// TIA Portal project "Project_IOLINKSafety" (V18)

(* hardware
DEVICE "S7-1200 station_1"  S7-1200 Station
   slot 0: "Rack_0"  S7-1200 Rack  Rack  V1.0
   slot 1: "PLC_1"  CPU 1212FC DC/DC/DC  6ES7 212-1AF40-0XB0  V4.6
DEVICE "GSD device_1"  GSD.Device.PN
   slot 0: "Rack"  Rack  V1.0
   slot 0: "AXL-F-BK-PN-TPS"  AXL F BK PN TPS  2403869  1.32
      slot 0: "AXL F BK PN TPS"  AXL F BK PN TPS
      slot 1: "Interface"  Interface
         slot 1: "RJ45 10/100 MBit/s"  RJ45 10/100 MBit/s
         slot 2: "RJ45 10/100 MBit/s_1"  RJ45 10/100 MBit/s
   slot 1: "AXL SE DI16/1_1"  AXL SE DI16/1  1088127  1.0
      slot 0: "AXL SE DI16/1"  AXL SE DI16/1
   slot 1: "Digital Input"  Digital Input
   slot 1: "AXL E IOL SDI8 SDO4 2A M12 6P PS2.4"  AXL E IOL SDI8 SDO4 2A M12 6P PS2.4
   slot 1: "AXL E IOL SDI8 SDO4 2A M12 L PS2.6"  AXL E IOL SDI8 SDO4 2A M12 L PS2.6
   slot 2: "AXL SE DO16/1_1"  AXL SE DO16/1  1088129  1.0
      slot 0: "AXL SE DO16/1"  AXL SE DO16/1
   slot 2: "Digital Input_1"  Digital Input
   slot 2: "Digital Input_1"  Digital Input
   slot 2: "Inactive_1"  Inactive
   slot 3: "AXL SE AI4 U 0-10_1"  AXL SE AI4 U 0-10  1088104  1.0
      slot 0: "AXL SE AI4 U 0-10"  AXL SE AI4 U 0-10
   slot 3: "Digital Input_2"  Digital Input
   slot 3: "Digital Input_2"  Digital Input
   slot 3: "Inactive"  Inactive
   slot 4: "AXL SE IOL4_1"  AXL SE IOL4  1088132  1.0
      slot 0: "AXL SE IOL4"  AXL SE IOL4
   slot 4: "Digital Input_3"  Digital Input
   slot 4: "Digital Input_3"  Digital Input
   slot 4: "Inactive_2"  Inactive
   slot 5: "Digital Input_4"  Digital Input
   slot 5: "Digital Input_4"  Digital Input
   slot 6: "Digital Input_5"  Digital Input
   slot 6: "Digital Input_5"  Digital Input
   slot 7: "Digital Input_6"  Digital Input
   slot 7: "Digital Input_6"  Digital Input
   slot 8: "Digital Input_7"  Digital Input
   slot 8: "Digital Input_7"  Digital Input
DEVICE "GSD device_2"  GSD.Device.PN
   slot 0: "Rack"  Rack  V1.0
   slot 0: "AXL-F-BK-PN-TPS_1"  AXL F BK PN TPS  2403869  1.32
      slot 0: "AXL F BK PN TPS"  AXL F BK PN TPS
      slot 1: "Interface"  Interface
         slot 1: "RJ45 10/100 MBit/s"  RJ45 10/100 MBit/s
         slot 2: "RJ45 10/100 MBit/s_1"  RJ45 10/100 MBit/s
   slot 1: "AXL SE DI16/1_1"  AXL SE DI16/1  1088127  1.0
      slot 0: "AXL SE DI16/1"  AXL SE DI16/1
   slot 1: "AXL E IOL SDI8 SDO4 2A M12 L PS2.6"  AXL E IOL SDI8 SDO4 2A M12 L PS2.6
   slot 2: "AXL SE DO16/1_1"  AXL SE DO16/1  1088129  1.0
      slot 0: "AXL SE DO16/1"  AXL SE DO16/1
   slot 2: "Digital Input"  Digital Input
   slot 3: "AXL SE AI4 U 0-10_1"  AXL SE AI4 U 0-10  1088104  1.0
      slot 0: "AXL SE AI4 U 0-10"  AXL SE AI4 U 0-10
   slot 3: "Digital Input_1"  Digital Input
   slot 4: "AXL SE IOL4_1"  AXL SE IOL4  1088132  1.0
      slot 0: "AXL SE IOL4"  AXL SE IOL4
   slot 4: "Digital Input_2"  Digital Input
*)

// ===== PLC "PLC_1"  CPU 1212FC DC/DC/DC =====
// protected blocks, not shown: "PRSF_AXL_E", "PRSF_DiagHandler", "PRSF_IOLM_Diag"

VAR_GLOBAL   // PLC tag table "Default tag table"
   "xActivate" AT %M0.0 : Bool;
   "Tag_1" AT %MW10 : Word;
   "Tag_2" AT %M0.1 : Bool;
   "Tag_3" AT %M0.2 : Bool;
   "Tag_4" AT %M0.3 : Bool;
   "mReset" AT %M1.3 : Bool;
   "Tag_6" AT %IW3 : Word;
   "Tag_7" AT %IW4 : Word;
   "Tag_8" AT %IW5 : Word;
   "Tag_9" AT %IW6 : Word;
   "Tag_10" AT %IW7 : Word;
   "Tag_11" AT %IW8 : Word;
   "Tag_12" AT %IW9 : Word;
   "Tag_13" AT %IW10 : Word;
   "Tag_14" AT %M1.4 : Bool;
   "siESTOP" AT %I3.0 : Bool;
   "sqESTOP1_Q" AT %Q3.0 : Bool;
END_VAR

TYPE "PRSF_UDT_IOCALL"
VERSION : 0.1
   STRUCT
      xReq : Bool;
      wHWAddr : Word;
      diCAP : DInt;
      xRDWR : Bool;
      iPort : Int;
      iIndex : Int;
      iSubindex : Int;
      iLen : Int;
      arr_b_IOLData : Array[0..231] of Byte;
      xDone_Valid : Bool;
      xBusy : Bool;
      xError : Bool;
      dwStatus : DWord;
      dwIOL_Status : DWord;
      iRD_Len : Int;
   END_STRUCT;
END_TYPE

TYPE "PRSF_UDT_DIAG"
VERSION : 0.1
   STRUCT
      wDiagCode : Word;
      wAddDiagCode : Word;
      xError : Bool;
      iState : Int;
      IOL_CallDiag : "PRSF_UDT_IOCALL";
   END_STRUCT;
END_TYPE

TYPE "PRSF_UDT_COM"
VERSION : 0.1
   STRUCT
      arr_i_Com : Array[0..255] of UInt;
      arr_HW : Array[0..8] of HW_ANY;
      arr_HW_Diag : Array[0..8] of Bool;
   END_STRUCT;
END_TYPE

DATA_BLOCK "Main_Safety_RTG1_DB"   // DB1, F_DB
{ S7_Optimized_Access := 'TRUE' }
NAME : FUSI
VERSION : 0.1
// stored: InstanceOfName Main_Safety_RTG1
"Main_Safety_RTG1"
BEGIN
END_DATA_BLOCK

DATA_BLOCK "PRSF_AXLE_UserDB"   // DB2
{ S7_Optimized_Access := 'TRUE' }
VERSION : 0.1
   VAR
      xActivate : Bool;
   END_VAR
   VAR RETAIN
      iPort : Int;
      IOLD_HWAddr : Hw_Any;
      IOLM_HWAddr : Hw_Any;
   END_VAR
   VAR
      wFAddr : Word;
      xSetFAddr : Bool;
      xErrorAck : Bool;
      wDevFAddr : Word;
      strDevSerial : String[13];
      xDiagAvailable : Bool;
      stDiagState : Struct
         uiLfdNo : UInt;
         uiPrio : UInt;
         bChannel : Byte;
         wCode : Word;
         FunctionGorup : String[8];
         dwAddValue : DWord;
         uiTextLength : UInt;
         strText : String[100];
      END_STRUCT;
      udtDiag : "PRSF_UDT_DIAG";
   END_VAR
BEGIN
END_DATA_BLOCK

DATA_BLOCK "Data_block_1"   // DB6
{ S7_Optimized_Access := 'TRUE' }
VERSION : 0.1
   VAR
      bytes : Array[0..999] of Byte;
   END_VAR
BEGIN
END_DATA_BLOCK

DATA_BLOCK "PRSF_AXL_E_COM"   // DB3200
{ S7_Optimized_Access := 'TRUE' }
VERSION : 0.1
   VAR
      udtCom : "PRSF_UDT_COM";
   END_VAR
BEGIN
END_DATA_BLOCK

FUNCTION_BLOCK "Main_Safety_RTG1"   // FB1, F_FBD
{ S7_Optimized_Access := 'TRUE' }
   VAR
      ACK_GL_Instance : ACK_GL;
      ESTOP1 : ESTOP1;
   END_VAR
   VAR CONSTANT
      OFF : Bool;
      ON : Bool := 1;
   END_VAR
BEGIN

REGION Network 1
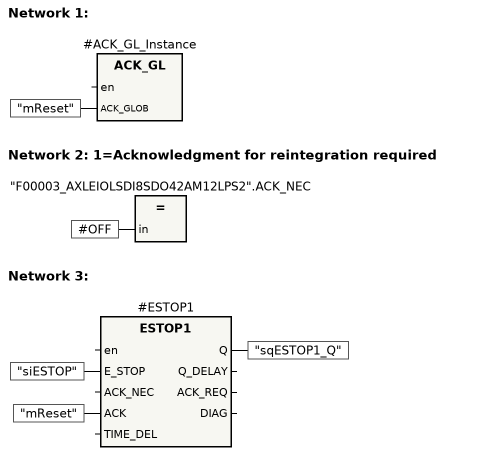
   #ACK_GL_Instance(ACK_GLOB := "mReset");   // ACK_GL
END_REGION

REGION Network 2: 1=Acknowledgment for reintegration required
   "F00003_AXLEIOLSDI8SDO42AM12LPS2".ACK_NEC := #OFF;
END_REGION

REGION Network 3
   #ESTOP1(E_STOP := "siESTOP", ACK := "mReset", Q => "sqESTOP1_Q");   // ESTOP1
END_REGION
END_FUNCTION_BLOCK

FUNCTION_BLOCK "IO_LINK_DEVICE"   // FB50001, SCL
TITLE = IO_LINK_DEVICE
{ S7_Optimized_Access := 'TRUE' }
AUTHOR : SUP_FA
FAMILY : IO-Link
VERSION : 3.0
// Function block to read and write acyclic data on devices with IO-Link used on SIMATIC S7 controllers. (former IO_LINK_CALL)
   VAR_INPUT
      REQ : Bool;   // Request Function / Neuer Auftrag / request function
      ID : Hw_Io;   // Hardwarekennung des IOL-Master Moduls (HW_IO) aus HW-Konfiguration / hardware identifier of IO-Link master module (HW_IO) from hw-config
      CAP : DInt := DINT#0;   // Client Access Point (CAP), bei ET200 immer 227 dez / Client Access Point (CAP), for ET200 always 227 decimal
      RD_WR : Bool;   // Lese und Schreibzugriff auf IO-Link Device 0: Lesen, 1: schreiben / read and write access on IO-Link device 0: read, 1: write
      PORT : Int := INT#0;   // Port/ Kanalnummer an dem das IO-Link Device betrieben wird. (ET200 = 0 .. 4) / number of port on IO-Link master module (ET200SP = 0..4)
      IOL_INDEX : Int := INT#0;   // Adressparameter Index (IO-Link Device) 0..32767 IOL-D, 65535 port functions / address parameter Index (IO-Link Device) 0..32767 IOL-D, 65535 port functions
      IOL_SUBINDEX : Int := INT#0;   // Adressparameter Subindex (IO-Link Device) 0 ges. Record; 1-255 einz. Parameter / address parameter Subindex (IO-Link Device) 0 full record; 1-255 single parameter
      LEN : Int := INT#0;   // Länge der zu schreibenden Daten (Nettodaten) / length of writing data (netto data)
   END_VAR
   VAR_OUTPUT
      DONE_VALID : Bool;   // Gültigkeit 0: Daten nicht gültig; 1: Daten gültig / validity 0: data invalid ; 1: data valid
      BUSY : Bool;   // 0: Auftrag abgeschlossen 1: Auftrag in Bearbeitung / 0: request finish 1: request in progress
      ERROR : Bool;   // Fehler Flag 0: kein Fehler; 1: Abbruch der Funktion mit Fehler / Error Flag = 0: no error; 1: function aborted with error
      STATUS : DWord := DW#16#00000000;   // DP/ PNIO - Fehlerstatus; ERROR Flag = 1 - detaillierter Kommunikationsfehlerstatus / DP/ PNIO - error status ; ERROR Flag = 1 - communication error status in detail
      IOL_STATUS : DWord := DW#16#00000000;   // IO-Link Fehlerstatus; ERROR Flag = 1 - detaillierte IO-Link Fehlerstatus / IO-Link error status; ERROR flag = 1: IO-Link error status in detail
      RD_LEN : Int := INT#0;   // Länge des gelesenen Datensatzes (Anzahl Bytes) / length of read data record (number of bytes)
   END_VAR
   VAR_IN_OUT
      RECORD_IOL_DATA : Array[0..231] of Byte;   // Datenbereich für LESEN / SCHREIBEN (max. 232 Byte) / data area for reading / writing data (max. 232 byte)
   END_VAR
   VAR
      RDREC_Function : RDREC;   // Funktion Datensatz lesen (ehemals SFB52) / system function "read data record" (former SFB52)
      WRREC_Function : WRREC;   // Funktion Datensatz schreiben (ehemals SFB53) / system function "write data record" (former SFB53)
      TP_poll : TP_TIME;   // Pollzeit für "Datensatz lesen" / poll rate read data record
      TON_monitoring : TON_TIME;   // Überwachungszeit für Aufträge / request monitoring time
      rdrec : Struct   // interne Struktur für RDREC / internal structure for RDREC
         valid : Bool;   // Function performed
         busy : Bool;   // Function busy
         error : Bool;   // Error flag
         status : DWord;   // Function result/error message
         length : UInt;   // Length of the fetched data record
      END_STRUCT;
      wrrec : Struct   // interne Struktur für WRREC / internal structure for WRREC
         length : UInt;   // length of write data record
         done : Bool;   // Function performed
         busy : Bool;   // Function busy
         error : Bool;   // Error flag
         status : DWord;   // Function result/error message
      END_STRUCT;
      read : Struct   // Datenbereich für Lesedaten / data area for reading data
         header : Struct
            CALL : Struct   // header for read/write data record
               Extended_Function_Num : Byte := 16#8;   // extended function number (fix coded 08h)
               Port : Byte;   // variable port (user interface) 0...255
               FI_Index : Word := 16#FE4A;   // FI index (fix coded 65098)
            END_STRUCT;
            IOL : Struct   // header for IO-Link
               Control : Byte;   // RD_WR = 0 = read = Control:=0x03 / / RD_WR = 1 = write = Control:=0x02
               Index_HighByte : Byte;   // index of data record 0…32767 (high byte)
               Index_LowByte : Byte;   // index of data record 0…32767 (low byte)
               Subindex : Byte;   // subindex for data record 0...255
            END_STRUCT;
         END_STRUCT;
         data : Array[0..231] of Byte;
      END_STRUCT;
      write : Struct   // Datenbereich für Schreibdaten / data area for writing data
         header : Struct
            CALL : Struct   // header for read/write data record
               Extended_Function_Num : Byte := 16#8;   // extended function number (fix coded 08h)
               Port : Byte;   // variable port (user interface) 0...255
               FI_Index : Word := 16#FE4A;   // FI index (fix coded 65098)
            END_STRUCT;
            IOL : Struct   // header for IO-Link
               Control : Byte;   // RD_WR = 0 = read = Control:=0x03 / / RD_WR = 1 = write = Control:=0x02
               Index_HighByte : Byte;   // index of data record 0…32767 (high byte)
               Index_LowByte : Byte;   // index of data record 0…32767 (low byte)
               Subindex : Byte;   // subindex for data record 0...255
            END_STRUCT;
         END_STRUCT;
         data : Array[0..231] of Byte;
      END_STRUCT;
      sequencecontrol : Int := INT#0;   // number of sequence control
      typeofrequest : Int := INT#0;   // type of request (0=Read, 1=Write)
      R_TRIG_REQ : Bool;   // Impuls für neuen Auftrag starten / impulse start new request
      R_TRIG_REQ_old : Bool;   // Flankenmerker / old value of REQ (previous cycle)
      F_TRIG_poll : Bool;   // Impuls für Pollen "Datensatz lesen" / impulse poll read data record (response)
      F_TRIG_poll_old : Bool;   // Flankenmerker / old value of Poll (previous cycle)
   END_VAR
   VAR_TEMP
      retval : Int;   // Variable für Rückgabewerte von Funktionen / function return value
      tmpWORD : Word;   // Datentyp WORD zur temporären Verwendung / data type WORD for temporarily use
      tmpDWORD : DWord;   // Datentyp DWORD zur temporären Verwendung / data type DWORD for temporarily use
      tmpINT : Int;   // Datentyp INT zur temporären Verwendung / data type INT for temporarily use
      i : Int;   // Laufvariable für for-Schleifen / run tag for counting loops
   END_VAR
BEGIN
   (*---------------------------------------------------------------------------------------------------------------------
   SIEMENS AG
   ©Copyright 2015. All Rights Reserved.
   -----------------------------------------------------------------------------------------------------------------------
   Limitation of liability
   This software was developed with largest care. However, the author can not guarantee, that the software runs under
   each version of STEP7 on each PLC flawlessly.
   There is no warranty for the software, to the extent permitted by applicable law. The copyright holder provides the
   software "as is" without warranty of any kind, either expressed or implied, including, but not limited to, the implied
   warranties of merchantability and fitness for a particular purpose. The entire risk as to the quality and performance
   of the software is with you. Should the software prove defective, you assume the cost of all necessary servicing,
   repair or correction. In no event unless required by applicable law will the copyright holder be liable to you for
   damages, including any general, special, incidental or consequential damages arising out of the use or inability to
   use the software (including but not limited to loss of data or data being rendered inaccurate or losses sustained by
   you or third parties or a failure of the software to operate with any other programs), even if such holder or other
   party has been advised of the possibility of such damages.
   Permission to use or copy this software for any purpose is hereby granted without fee, provided the above notices are
   retained on all copies. Permission to modify the code and to distribute modified code is granted, provided the above
   notices are retained, and a notice that the code was modified is included with the above copyright notice.
   -----------------------------------------------------------------------------------------------------------------------
   Functionality provided by this source (short description):
   Function block IO_LINK_DEVICE - used to read and write of acyclic data records on devices with IO-Link.
   Note:
   To read data records, the IO-Link master modules needs to know which data record is required. Therefore it is necessary
   to send at first a request via write data record (only header of 8 byte). As response the IO-Link master module
   will send the required data record.

   Status:     Released (tested)
   File name:  IO_LINK_DEVICE
   System :    SIMATIC S7-1200/1500
   Version :   3.1
   -----------------------------------------------------------------------------------------------------------------------
   Script to be stored on level ... in project (mark appropriate levels with [x] below)
   [ ] External
   [ ] All levels possible
   [x] Project level
   [ ] Controller level
   [ ] Device level
   [ ] Subobject level
   -----------------------------------------------------------------------------------------------------------------------
   Restrictions, known limitations:
   The limitation of 240 byte is based on PROFIBUS DP protocol. With PROFINET IO there wouldn't no limit but because of 
   compatibility reason it wasn't changed.
     - header =   8 byte
     - data   = 232 byte
   -----------------------------------------------------------------------------------------------------------------------
   Requirements, prerequisites, External resources used: nothing
   -----------------------------------------------------------------------------------------------------------------------
   Change log table (latest change is at the bottom OF the list):
   Version Date Changes applied
   V2.0.0 <2013-09-30> First created with TIA Portal V12 SP1
   V2.1.0 <2014-03-14> Upgrade system function 'WRREC' from V1.0 to V1.1 and released for TIA Portal V13
   V3.0.0 <2015-02-28> Upgrade and released for TIA Portal V13 SP1 (without backup/restore master parameter)
   V3.1.0 <2015-09-15> Change of #IOL_INDEX and #Port lower boundry to 0 and Improved behaviour when called in cyclic OBs with > 100ms
   ---------------------------------------------------------------------------------------------------------------------*)

   (*---------------------------------------------------------------------------------------------------------------------
   Description of programmed IO-Link error codes
   8000 = time out
   8001 = wrong port
   8002 = wrong index
   8003 = wrong subindex
   8005 = wrong length for write data record
   8006 = wrong length for read data record
   8052 = error during reading data record
   8053 = error during writing data record
   All other codes are coming from a higher level!
   ---------------------------------------------------------------------------------------------------------------------*)

   (*---------------------------------------------------------------------------------------------------------------------
               NEW REQUEST
   ---------------------------------------------------------------------------------------------------------------------*)
   // detection rising edge of "REQ"
   #R_TRIG_REQ := #REQ = TRUE AND #R_TRIG_REQ_old = FALSE;
   #R_TRIG_REQ_old := #REQ = TRUE;

   // start new request if not busy
   IF #R_TRIG_REQ = TRUE AND #sequencecontrol = 0 THEN
       // Freeze record ID and CAP
       #WRREC_Function.ID := #ID;
       #WRREC_Function.INDEX := #CAP;
       #RDREC_Function.ID := #ID;
       #RDREC_Function.INDEX := #CAP;

       // Initialize outputs
       #DONE_VALID := FALSE;
       #BUSY := TRUE;
       #ERROR := FALSE;
       #STATUS := DW#16#00000000;
       #IOL_STATUS := DW#16#00000000;
       #RD_LEN := INT#0;

       // Initialize data area
       #read.header."CALL"."Port" := B#16#0;
       #read.header.IOL.Index_LowByte := B#16#0;
       #read.header.IOL.Index_HighByte := B#16#0;
       #read.header.IOL.Subindex := B#16#0;
       #i := INT#0; // initialize loop counter      
       FOR #i := 0 TO 231 DO
           #write.data[#i] := B#16#0;
           #read.data[#i] := B#16#0;
       END_FOR;

   (*---------------------------------------------------------------------------------------------------------------------
       Setup IO-LINK Call needs a specific header
   ---------------------------------------------------------------------------------------------------------------------*)
   // setup CALL header
   #write.header."CALL".Extended_Function_Num := 16#08;  // extended function number (fix coded 08h)
   #write.header."CALL"."Port" := INT_TO_BYTE(#PORT);  // 1..63 = PORT number, 64..255=reserved
   #write.header."CALL".FI_Index := 65098;  // IOL-Header is following (fix coded 65098)

   // setup IOL header 
   // CONTROL = please see below at BODY
   // INDEX
   #write.header.IOL.Index_LowByte := INT_TO_BYTE(#IOL_INDEX);
   #tmpWORD := INT_TO_WORD(#IOL_INDEX);
   #tmpWORD := SHR(IN := #tmpWORD, N := 8);
   #write.header.IOL.Index_HighByte := WORD_TO_BYTE(#tmpWORD);
   // SUBINDEX
   #write.header.IOL.Subindex := INT_TO_BYTE(#IOL_SUBINDEX);

   // BODY (data max. 232 Byte, Array 0..231 of Byte) 
   IF #RD_WR = TRUE THEN
       // IO-Link write data record requested, copy data from "RECORD_IOL_DATA"
       #write.header.IOL.Control := B#16#02; // CONTROL B#16#02 = write data record
       #wrrec.length := INT_TO_UINT(#LEN) + UINT#8;  // data length header + data = IO-Link write data record
       #typeofrequest := 2; // write data record
       // copy IOL_RECORD_DATA in working area
       #i := INT#0;    // initialize loop counter 
       FOR #i := 0 TO #LEN - 1 DO
           #write.data[#i] := #RECORD_IOL_DATA[#i];
       END_FOR;
   ELSE
       // IO-Link read data record requested
       #write.header.IOL.Control := 16#03;  // CONTROL 16#03 = read data record
       #wrrec.length := UINT#8; // data length only header = IO-Link read data record
       #typeofrequest := 1; // read data record        
   END_IF;
   #sequencecontrol := 1;  // Start sequence
   ELSE
       ;
   END_IF;

   (*---------------------------------------------------------------------------------------------------------------------
               SEQUENCE CONTROL
   ---------------------------------------------------------------------------------------------------------------------*)
   CASE #sequencecontrol OF
       1:  // Check input parameter        
           IF #PORT < INT#0 OR #PORT > INT#63 THEN // PORT (Wrong port address = 0x8001)
               #ERROR := TRUE;
               #IOL_STATUS := DW#16#80010000;
               #sequencecontrol := 99; // aborting function with error
           ELSIF #IOL_INDEX < INT#0 OR #IOL_INDEX > INT#32767 THEN    // INDEX (Wrong index = 0x8002)
               #ERROR := TRUE;
               #IOL_STATUS := DW#16#80020000;
               #sequencecontrol := 99; // aborting function with error
           ELSIF #IOL_SUBINDEX < INT#0 OR #IOL_SUBINDEX > INT#255 THEN    // SUBINDEX (Wrong subindex = 0x8003)
               #ERROR := TRUE;
               #IOL_STATUS := DW#16#80030000;
               #sequencecontrol := 99; // aborting function with error
           ELSIF #typeofrequest = 2 AND (#LEN < 1 OR #LEN > 232) THEN  // LEN (wrong length for write data record = 0x8004)
               #ERROR := TRUE;
               #IOL_STATUS := DW#16#80050000;
               #sequencecontrol := 99; // aborting function with error
           ELSIF #typeofrequest = 1 AND (#LEN < 0 OR #LEN > 232) THEN  // LEN (wrong length for read data record = 0x8005)
               #ERROR := TRUE;
               #IOL_STATUS := DW#16#80060000;
               #sequencecontrol := 99; // aborting function with error
           ELSE    // all input parameter are right
               #sequencecontrol := 2;
           END_IF;

       2:  (*-------------------------------------------------------------------------------------------------------------
           WRREC = Write Data Record
           Note:
           To read data records, the IO-Link master modules needs to know which PORT is required. Therefore it is necessary
           to send at first a request via write data record (header, 8 byte). As response the IO-Link master module will 
           send the required data record.
           -------------------------------------------------------------------------------------------------------------*)
           #WRREC_Function(REQ := TRUE,
                           LEN := #wrrec.length,
                           DONE => #wrrec.done,
                           BUSY => #wrrec.busy,
                           ERROR => #wrrec.error,
                           STATUS => #wrrec.status,
                           RECORD := #write);
           // output status during write data record
           IF #wrrec.busy THEN
               #STATUS := #wrrec.status;
               #IOL_STATUS := DW#16#00020000;  // 0002 = writing in progress 
           ELSIF #wrrec.error THEN
               #tmpDWORD := #wrrec.status AND DW#16#00FFFF00;  // filter status
               IF #tmpDWORD = DW#16#0080C200 THEN    // if resource #BUSY (#STATUS=80C2), then ... 
                   #sequencecontrol := 3;  // ... repeat write data record
               ELSE
                   #ERROR := TRUE;
                   #STATUS := #wrrec.status;   // ... otherwise output error status of "WRREC"
                   #IOL_STATUS := DW#16#80530000;  // ... with note '8053' = error status of "WRREC"
                   #sequencecontrol := 99; // aborting function with error
               END_IF;
           ELSIF #wrrec.done = TRUE THEN   // wait for write data record finish without error
               #TP_poll(IN := TRUE,
                        PT := T#100ms);    // poll for response
               #F_TRIG_poll_old := #TP_poll.Q = TRUE;  // save old value for neg edge detection independant of pulse time

               #sequencecontrol := 4;
           ELSE
               ;
           END_IF;

       3:  // repeat write data record because resource was busy
           #WRREC_Function(REQ := FALSE);
           #sequencecontrol := 2;

       4:  // wait and poll for response = Read Data Record (RDREC)
           #WRREC_Function(REQ := FALSE);
           #TP_poll(IN := TRUE,
                    PT := T#100ms);

           // if poll rate executed then start read data record (on falling edge)
           #F_TRIG_poll := #TP_poll.Q = FALSE AND #F_TRIG_poll_old = TRUE;
           #F_TRIG_poll_old := #TP_poll.Q = TRUE;

           // RDREC = Read Data Record
           #RDREC_Function(REQ := #F_TRIG_poll,
                           MLEN := UINT#0, // length = 0 = read all data which are available
                           VALID => #rdrec.valid,
                           BUSY => #rdrec.busy,
                           ERROR => #rdrec.error,
                           STATUS => #rdrec.status,
                           LEN => #rdrec.length,
                           RECORD := #read);
           // output status during read data record
           IF #rdrec.busy THEN
               #STATUS := #rdrec.status;
               #IOL_STATUS := DW#16#00030000; // 16#0003 = reading in progress
           ELSIF #rdrec.error = TRUE THEN
               #tmpDWORD := #rdrec.status AND DW#16#00FFFF00;  // filter status
               IF #tmpDWORD = DW#16#0080C200 THEN  // if resource busy (status=80C2), then ... 
                   #sequencecontrol := 5;  // ... repeat read data record / continue polling
               ELSE
                   #ERROR := TRUE;
                   #STATUS := #rdrec.status;   // ... otherwise output error code of "RDREC"
                   #IOL_STATUS := DW#16#80520000;  // ... with note '8052' = error status of "RDREC"
                   #sequencecontrol := 99; // aborting function with error
               END_IF;
           ELSIF #rdrec.valid THEN
               IF  // check the response wether it matches the request (compare PORT, INDEX and SUBINDEX)
                   (#write.header."CALL"."Port" <> #read.header."CALL"."Port") OR
                   (#write.header.IOL.Index_HighByte <> #read.header.IOL.Index_HighByte) OR
                   (#write.header.IOL.Index_LowByte <> #read.header.IOL.Index_LowByte) OR
                   (#write.header.IOL.Subindex <> #read.header.IOL.Subindex)
               THEN    // read data record don't match the request
                   #ERROR := TRUE;
                   #STATUS := #rdrec.status;
                   #IOL_STATUS := DW#16#70000000;  // output status '7000', no consistent data
                   #sequencecontrol := 99; // aborting function with error
               ELSIF #read.header.IOL.Control = B#16#80 THEN   // check the response for IO-Link errors
                   // State 0x80 = IOL_CALL_RES PDU shows IO-Link error detect
                   #ERROR := TRUE;
                   #STATUS := DW#16#00000000;
                   #IOL_STATUS.%B3 := #read.data[0];   // IO-Link master error code
                   #IOL_STATUS.%B2 := #read.data[1];   // IO-Link master error code
                   #IOL_STATUS.%B1 := #read.data[2];  // IO-Link device error code
                   #IOL_STATUS.%B0 := #read.data[3];  // IO-Link device additional error code

                   #sequencecontrol := 99; // aborting function with error
               ELSE    // read data are valid = output
                   #DONE_VALID := TRUE;
                   #BUSY := FALSE;
                   #ERROR := FALSE;
                   #STATUS := DW#16#00000000;
                   #IOL_STATUS := DW#16#00000000;  // request finished

                   IF #typeofrequest = 1 THEN
                       #RD_LEN := UINT_TO_INT(#rdrec.length - UINT#8);  // device parameter cover header and data,
                       // only data will be output
                       #i := INT#0; // initialize loop counter
                       FOR #i := 0 TO UINT_TO_INT(#rdrec.length - UINT#8 - UINT#1) DO
                           #RECORD_IOL_DATA[#i] := #read.data[#i];
                       END_FOR;
                   ELSE
                       ;
                   END_IF;
                   #sequencecontrol := 98;
               END_IF;
           ELSE
               ;
           END_IF;

       5:  // poll again for response because resource was busy
           #TP_poll(IN := FALSE,
                    PT := T#100ms);
           #RDREC_Function(REQ := FALSE,
                           RECORD := #read);
           #sequencecontrol := 4;  // ... repeat read data record / continue polling   

       98: // request done successfully
           #TP_poll(IN := FALSE,
                    PT := T#100ms);
           #RDREC_Function(REQ := FALSE,
                           RECORD := #read);
           IF #REQ = FALSE THEN
               #DONE_VALID := FALSE;
               #BUSY := FALSE;
               #ERROR := FALSE;
               #RD_LEN := INT#0;
               #STATUS := DW#16#00000000;
               #IOL_STATUS := DW#16#00010000; // ready for new request
               #sequencecontrol := 0;
               #typeofrequest := 0;
           ELSE
               ;
           END_IF;

       99: // Function aborted with error
           #TP_poll(IN := FALSE,
                    PT := T#100ms);
           #WRREC_Function(REQ := FALSE);
           #RDREC_Function(REQ := FALSE,
                           RECORD := #read);
           #DONE_VALID := FALSE;
           #BUSY := FALSE;
           #RD_LEN := INT#0;
           #sequencecontrol := 0;
           #typeofrequest := 0;

       ELSE  // no relevant case, ready for new request
           #WRREC_Function(REQ := FALSE);
           #RDREC_Function(REQ := FALSE,
                           RECORD := #read);
           #TP_poll(IN := FALSE,
                    PT := T#100ms);
           #TON_monitoring(IN := FALSE,
                           PT := T#20s);
           #sequencecontrol := 0;
           #typeofrequest := 0;
   END_CASE;

   (*---------------------------------------------------------------------------------------------------------------------
               MONITORING
   ---------------------------------------------------------------------------------------------------------------------*)
   #TON_monitoring(IN := #sequencecontrol > 0 AND #sequencecontrol < 98,
                   PT := T#20s);
   IF #TON_monitoring.Q THEN
       #ERROR := TRUE;
       #IOL_STATUS := DW#16#80000000; // request time out       
       #sequencecontrol := 99; // aborting function with error
   END_IF;
END_FUNCTION_BLOCK

ORGANIZATION_BLOCK "Main"   // OB1, LAD, ProgramCycle
TITLE = "Main Program Sweep (Cycle)"
{ S7_Optimized_Access := 'TRUE' }
VERSION : 0.1
   VAR_INPUT
      Initial_Call : Bool;   // Initial call of this OB
      Remanence : Bool;   // =True, if remanent data are available
   END_VAR
BEGIN
END_ORGANIZATION_BLOCK

ORGANIZATION_BLOCK "Cyclic interrupt"   // OB30, FBD, CyclicInterrupt
{ S7_Optimized_Access := 'TRUE' }
VERSION : 0.1
   VAR_INPUT
      Initial_Call : Bool;   // Initial call of this OB
      Event_Count : Int;   // Events discarded
   END_VAR
BEGIN

REGION Network 2
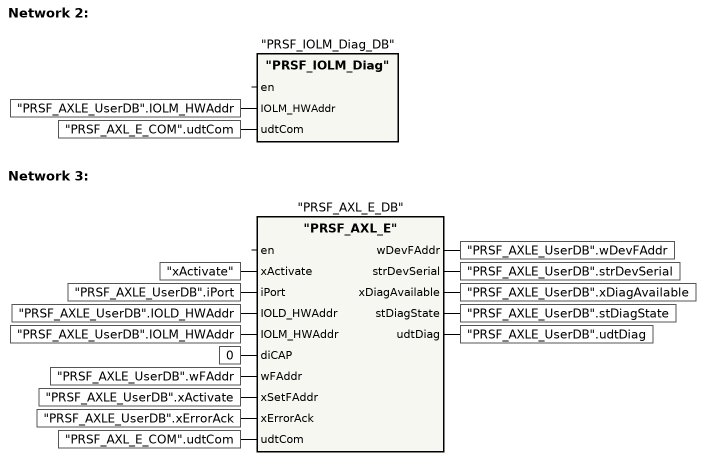
   "PRSF_IOLM_Diag_DB"(IOLM_HWAddr := "PRSF_AXLE_UserDB".IOLM_HWAddr, udtCom := "PRSF_AXL_E_COM".udtCom);   // "PRSF_IOLM_Diag"
END_REGION

REGION Network 3
   "PRSF_AXL_E_DB"(xActivate := "xActivate",   // "PRSF_AXL_E"
                   iPort := "PRSF_AXLE_UserDB".iPort,
                   IOLD_HWAddr := "PRSF_AXLE_UserDB".IOLD_HWAddr,
                   IOLM_HWAddr := "PRSF_AXLE_UserDB".IOLM_HWAddr,
                   diCAP := 0,
                   wFAddr := "PRSF_AXLE_UserDB".wFAddr,
                   xSetFAddr := "PRSF_AXLE_UserDB".xActivate,
                   xErrorAck := "PRSF_AXLE_UserDB".xErrorAck,
                   udtCom := "PRSF_AXL_E_COM".udtCom,
                   wDevFAddr => "PRSF_AXLE_UserDB".wDevFAddr,
                   strDevSerial => "PRSF_AXLE_UserDB".strDevSerial,
                   xDiagAvailable => "PRSF_AXLE_UserDB".xDiagAvailable,
                   stDiagState => "PRSF_AXLE_UserDB".stDiagState,
                   udtDiag => "PRSF_AXLE_UserDB".udtDiag);
END_REGION
END_ORGANIZATION_BLOCK